# EPICS autosave request: iocs/XSPDIOC/iocBoot/iocXSPD/auto_settings.req
file "ADXSPD_settings.req",  P=$(P),  R=cam1:
file "NDStdArrays_settings.req",  P=$(P),  R=image1:
file "commonPlugin_settings.req", P=$(P)
